FUNCTION_BLOCK Comp_Send_Receive (* Basic Function Block Type *)
  (* Standard: 61499-2 *)
  (* Version 0.0, 25/02/2022, SESA197029, Template *)
  PACKAGE SE.Nereda;
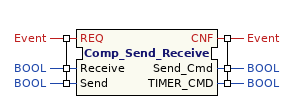
  EVENT_INPUT
    REQ WITH Receive, Send; (* Normal Execution Request *)
  END_EVENT
  EVENT_OUTPUT
    CNF WITH Send_Cmd, TIMER_CMD; (* Execution Confirmation *)
  END_EVENT
  VAR_INPUT
    Receive : BOOL; (* Input event qualifier *)
    Send : BOOL;
  END_VAR
  VAR_OUTPUT
    Send_Cmd : BOOL := TRUE; (* Output event qualifier *)
    TIMER_CMD : BOOL;
  END_VAR
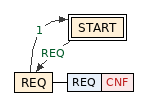
  EC_STATES
    START; (* Initial State *)
    REQ : REQ -> CNF; (* Normal execution *)
  END_STATES
  EC_TRANSITIONS
    START TO REQ := REQ;
    REQ TO START := 1;
  END_TRANSITIONS
  ALGORITHM REQ IN ST: (* Normally executed algorithm *)
IF Send=Receive AND Send=TRUE THEN
	Send_Cmd:=FALSE;
END_IF;

IF Send=Receive AND Send=FALSE THEN
	Send_Cmd:=TRUE;
END_IF;

IF Send<>Receive THEN
	TIMER_CMD:=TRUE;
ELSE
	TIMER_CMD:=FALSE;
END_IF;
;
  END_ALGORITHM
END_FUNCTION_BLOCK
